PROGRAM MAIN
VAR
	mqtt: MQTT;
	
	tonTimer : TON := (PT:=T#1S); //Interval timer for broadcasting.
	counter : INT := 0;
	isPublished : BOOL := FALSE;
END_VAR

IF _TaskInfo[GETCURTASKINDEXEX()].FirstCycle THEN
	mqtt.configureMQTTClient();
END_IF 
mqtt.connect();

IF mqtt.isConnected() THEN
	//Capasity test
	IF NOT isPublished THEN
		mqtt.publish(msg := 'this is a very long message for testing mqtt maximum capacity. this is a very lo');
		isPublished := TRUE;
	END_IF

	
	
    //tonTimer(IN:=TRUE);
    //IF tonTimer.Q THEN
		//msg test
		//mqtt.publish(msg := '{"temperature":345;"motorSpeed":300;"distance":1345;"humidity":58}');
	
	
		//counter test
		//counter := counter + 1;		
        //tonTimer(IN:=FALSE);  
        //mqtt.publish(msg := TO_STRING(counter));
    //END_IF
	
END_IF

END_PROGRAM

(* stored: Version 1.1.0.1, ProductVersion 3.1.4024.12
   POU MAIN: Id {bcad94f3-26d4-4398-99c6-2ab4d243b808}, SpecialFunc None *)
